FUNCTION_BLOCK PLC2Communicaton
VAR_INPUT
END_VAR
VAR_OUTPUT
END_VAR
VAR
END_VAR

END_FUNCTION_BLOCK

(* stored: Version 1.1.0.1, ProductVersion 3.1.4024.13
   POU PLC2Communicaton: Id {9a88c0eb-c600-4a7f-b81d-78081ad1ee13}, SpecialFunc None *)
